(* IEC 61131-3 sources: LMM/plc, 1 file *)

(* ---- GVL.st ---- *)
VAR_GLOBAL
(* =========================================================================
   LMM 拉毛机 全局变量（唯一 GVL）
   轴：X=M1+M2，Y=M3，Z=M4，R=M5。跨距 = Y 行程（HMI_rWheelBase，4~6 m）。
   维护方式：编辑本文件后运行 tools/inject_st.py 注入 LMM.xml。
   ========================================================================= *)

(* ===== 1. 面板物理 IO（地址固定勿改） ===== *)
StartBtn AT %IX1.6 : BOOL;      (* 【面板启动】→ HMI_xStart *)
StopBtn AT %IX1.4 : BOOL;       (* 【面板停止】→ HMI_xStop *)
ResetBtn : BOOL;                (* 【面板复位】→ HMI_xStopHold3s；地址现场另绑 *)
EStop AT %IX0.4 : BOOL;         (* 【面板急停】正常=TRUE 按下=FALSE *)
StopLamp AT %QX0.6 : BOOL;      (* 【停止指示灯】← Dev_xStop *)
StartLamp AT %QX0.7 : BOOL;     (* 【运行指示灯】← Dev_xRun *)
JogFwd : BOOL;                  (* 【面板前进】手动 X+ *)
JogBwd : BOOL;                  (* 【面板后退】手动 X- *)
JogRight : BOOL;                (* 【面板右】手动 Y+ *)
JogLeft : BOOL;                 (* 【面板左】手动 Y- *)
JogUp : BOOL;                   (* 【面板上】手动 Z+ *)
JogDown : BOOL;                 (* 【面板下】手动 Z- *)
JogClockAdd : BOOL;             (* 【面板顺时针】手动 R+ *)
JogClockMis : BOOL;             (* 【面板逆时针】手动 R- *)

(* ===== 2. 安全 / 起停（PRG_TcpHmi 仲裁后写） ===== *)
HMI_xEStop : BOOL;              (* 【急停】TRUE正常 FALSE按下 = 物理 AND 触摸屏Req AND Web *)
HMI_xStop : BOOL;               (* 【停止】任一源为真即停；长按3s=复位 *)
HMI_xStopHold3s : BOOL;         (* 【复位】清急停锁存 + 轴故障复位 *)
HMI_xStart : BOOL;              (* 【启动】上升沿 *)
HMI_xEnable : BOOL;             (* 【启动别名】与 HMI_xStart 等效 *)
xEStopLatched : BOOL;           (* 【急停锁存】仅复位可清 *)
xFaultAggregate : BOOL;         (* 【故障汇总】任轴 ErrorStop *)
eCtrlSrc : INT;                 (* 【控制源】0=面板/触摸屏 1=远程Web；仅 PRG_TcpHmi 写 *)

(* ===== 3. 设备状态显示（Logic 写，只读派生，不做互锁） ===== *)
eOpMode : INT;                  (* 【运行方式】0手动 1自动 *)
iAlarmID : INT;                 (* 【内部报警号】 *)
HMI_eDevState : INT;            (* 【只读·状态码】0停 1运行 2错误 *)
HMI_eOpMode : INT;              (* 【只读·方式显示】0手动 1自动 *)
HMI_iAlarmShow : INT;           (* 【只读·报警号】1001急停 1002轴故障 1005力超时 1006从站失败 1007未就绪；1008已废 *)
Dev_xStop : BOOL;               (* 【内部·停止派生】 *)
Dev_xRun : BOOL;                (* 【内部·运行派生】 *)
Dev_xError : BOOL;              (* 【内部·故障派生】 *)
HMI_xDevStop : BOOL;            (* 【只读·停止灯】 *)
HMI_xDevRun : BOOL;             (* 【只读·运行灯】 *)
HMI_xDevError : BOOL;           (* 【只读·故障灯】 *)
HMI_xLampEStop : BOOL;          (* 【只读·急停指示】 *)
HMI_xLampEnableOk : BOOL;       (* 【只读·就绪灯】 *)
HMI_xLampFault : BOOL;          (* 【只读·故障指示】 *)

(* ===== 4. 手动点动（电平；前提：急停正常+手动+未停止） ===== *)
HMI_xAutoMode : BOOL;           (* 【模式】FALSE手动 TRUE自动 *)
HMI_xJogXPos : BOOL;            (* 【X+】M1=M2 同速同向；与旋转互斥 *)
HMI_xJogXNeg : BOOL;            (* 【X-】 *)
HMI_xSpinLeft : BOOL;           (* 【左旋转】差速原地转；与 X± 互斥 *)
HMI_xSpinRight : BOOL;          (* 【右旋转】 *)
HMI_xJogYPos : BOOL;            (* 【Y+】受限位 *)
HMI_xJogYNeg : BOOL;            (* 【Y-】 *)
HMI_xJogZPos : BOOL;            (* 【Z+】回零后软限位 [-0.7,0] *)
HMI_xJogZNeg : BOOL;            (* 【Z-】 *)
HMI_xJogRPos : BOOL;            (* 【R+】需 xM5Ready *)
HMI_xJogRNeg : BOOL;            (* 【R-】 *)
(* 点动速度 HMI_rJogVel*/rSpinVel 在 RETAIN 区 *)

(* ===== 5. 回零（上升沿；同时只回一轴） ===== *)
HMI_xHomeY : BOOL;              (* 【Y回零】 *)
HMI_xHomeZ : BOOL;              (* 【Z回零】完成后软限位生效 *)
HMI_xHomeR : BOOL;              (* 【R回零】编码器回零 *)
HMI_iHomeAxis : INT := 0;       (* 【回零轴选择】0无 1Y 2Z 3R *)
HMI_xHomeExec : BOOL;           (* 【回零执行】对选定轴 *)
HMI_xHomedY : BOOL;             (* 【只读·Y已回零】 *)
HMI_xHomedZ : BOOL;             (* 【只读·Z已回零】 *)
HMI_xHomedR : BOOL;             (* 【只读·R已回零】 *)
HMI_xHomeBusyY : BOOL;          (* 【只读·Y回零中】 *)
HMI_xHomeBusyZ : BOOL;          (* 【只读·Z回零中】 *)
HMI_xHomeBusyR : BOOL;          (* 【只读·R回零中】 *)

(* ===== 6. 自动多道循环 ===== *)
HMI_xAutoStart : BOOL;          (* 【自动启动】上升沿 *)
HMI_xAutoAbort : BOOL;          (* 【自动中止】立即结束 *)
HMI_rHeadingErr : REAL := 0.0;  (* 【航向误差】视觉/外部纠偏输入（实时量，不保持） *)
iAutoStep : INT;                (* 【自动步】0Idle..6Done *)
HMI_iAutoStepShow : INT;        (* 【只读·自动步号】 *)
HMI_xAutoBusy : BOOL;           (* 【只读·自动忙】 *)
HMI_xAutoDone : BOOL;           (* 【只读·自动完成】 *)
(* 自动参数 rAutoDistX/rAutoVel*/rWheelBase/iAutoPasses/rKp*/rForceSet 在 RETAIN 区 *)

(* ===== 7. 力控（LE 拉压传感器，组态 Modbus RTU COM0） ===== *)
Force_xEnable : BOOL := TRUE;   (* 【力通讯总使能】 *)
Force_wInRaw AT %IW102 : WORD;  (* 组态读通道：0x0000 原始力 *)
Force_wOutTare AT %QW42 : WORD; (* 组态写通道：0x0011 去皮 *)
Force_wOutUnit AT %QW43 : WORD := 5; (* 组态写通道：0x0002 单位 5=N *)
Force_rScale : REAL := 0.01;    (* 原始值倍率 *)
Force_xReadTrig : BOOL;         (* 【内部·力读触发】组态用，勿绑屏 *)
Force_xCommOk : BOOL;           (* 【只读·力通讯正常】 *)
Force_xTimeout : BOOL;          (* 【只读·力超时】报警1005 *)
Force_xSlaveFail : BOOL;        (* 【只读·从站使能失败】报警1006 *)
Force_xTareBusy : BOOL;         (* 【只读·去皮中】 *)
Force_xTareDone : BOOL;         (* 【只读·去皮完成】 *)
Force_iRaw : INT;               (* 【只读·原始计数】 *)
Force_iState : INT;             (* 【只读·力任务状态】 *)
rForceAct : REAL;               (* 【实际力】N；Axis 任务写（模拟时 Logic 写） *)
rForceKp : REAL;                (* 【内部·恒力Kp】 *)
HMI_rForceSim : REAL;           (* 【力模拟值】N *)
HMI_xForceSimEnable : BOOL;     (* 【力模拟使能】台架用 *)
HMI_xForceTare : BOOL;          (* 【去皮】上升沿 *)
HMI_xForceUntare : BOOL;        (* 【取消去皮】上升沿 *)
HMI_xForceGuide : BOOL;         (* 【力引导电平】TRUE 持续 Z 恒力跟随 *)
HMI_rForceShow : REAL;          (* 【只读·显示力】N *)
Logic_xForceTare : BOOL;        (* 【内部·自动步去皮脉冲】 *)

(* ===== 8. 硬限位配置已移至 RETAIN 区（Cfg_rLim*） ===== *)

(* ===== 9. 联锁 / 物理限位输入（地址 TBD，设备树映射） ===== *)
I_xLimYPos : BOOL;              (* 【Y正限位开关】 *)
I_xLimYNeg : BOOL;              (* 【Y负限位开关】 *)
I_xLimZPos : BOOL;              (* 【Z正限位开关】 *)
I_xLimZNeg : BOOL;              (* 【Z负限位开关】 *)
xIlk_BlockYPlus : BOOL;         (* 【联锁禁Y+】开关 ∨ Cfg 限位 *)
xIlk_BlockYNeg : BOOL;          (* 【联锁禁Y-】 *)
xIlk_BlockZPlus : BOOL;         (* 【联锁禁Z+】 *)
xIlk_BlockZNeg : BOOL;          (* 【联锁禁Z-】 *)
xM5Ready : BOOL := TRUE;        (* 【第5轴就绪】FALSE=忽略 R *)

(* ===== 10. 轴命令（Logic → Axis，仅 Logic 写） ===== *)
AxisCmd_xPower : BOOL;          (* 【轴使能】= 安全条件 *)
AxisCmd_xStopAll : BOOL;        (* 【全停】急停/停止/故障/中止 *)
AxisCmd_xResetFault : BOOL;     (* 【故障复位脉冲】 *)
AxisCmd_xJogXPos : BOOL;        (* 【X+】 *)
AxisCmd_xJogXNeg : BOOL;        (* 【X-】 *)
AxisCmd_xSpinLeft : BOOL;       (* 【左旋】 *)
AxisCmd_xSpinRight : BOOL;      (* 【右旋】 *)
AxisCmd_xJogYPos : BOOL;        (* 【Y+】 *)
AxisCmd_xJogYNeg : BOOL;        (* 【Y-】 *)
AxisCmd_xJogZPos : BOOL;        (* 【Z+】 *)
AxisCmd_xJogZNeg : BOOL;        (* 【Z-】 *)
AxisCmd_xJogRPos : BOOL;        (* 【R+】 *)
AxisCmd_xJogRNeg : BOOL;        (* 【R-】 *)
AxisCmd_xHomeY : BOOL;          (* 【Y回零】完成/停止清 *)
AxisCmd_xHomeZ : BOOL;          (* 【Z回零】 *)
AxisCmd_xHomeR : BOOL;          (* 【R回零】 *)
AxisCmd_xMoveRelX : BOOL;       (* 【X相对走距】速度模式+里程判完成 *)
AxisCmd_rMoveDistX : REAL;      (* 【X相对距离】 *)
AxisCmd_rMoveVelX : REAL;       (* 【X相对速度】 *)
AxisCmd_xMoveRelY : BOOL;       (* 【Y相对】 *)
AxisCmd_rMoveDistY : REAL;      (* 【Y相对距离】自动=跨距 *)
AxisCmd_rMoveVelY : REAL;       (* 【Y速度】 *)
AxisCmd_xMoveAbsY : BOOL;       (* 【Y绝对】归位用 *)
AxisCmd_rMoveAbsPosY : REAL;    (* 【Y绝对目标】 *)
AxisCmd_xForceFollow : BOOL;    (* 【Z力跟随】 *)
AxisCmd_rForceSet : REAL;       (* 【力目标】 *)
AxisCmd_rForceKp : REAL;        (* 【力Kp】 *)
AxisCmd_rForceVelMax : REAL;    (* 【力跟随限速】 *)
AxisCmd_xHoldR : BOOL;          (* 【R保持角】 *)
AxisCmd_rRHoldPos : REAL;       (* 【R保持角位置】 *)
AxisCmd_rHeadingErr : REAL;     (* 【航向误差】 *)
AxisCmd_rTrackKp : REAL;        (* 【纠偏Kp】 *)
AxisCmd_rJogVelX : REAL;        (* 【X点动速度】 *)
AxisCmd_rSpinVel : REAL := 0.0; (* 【旋转速度】 *)
AxisCmd_rJogVelY : REAL;        (* 【Y点动速度】 *)
AxisCmd_rJogVelZ : REAL;        (* 【Z点动速度】 *)
AxisCmd_rJogVelR : REAL;        (* 【R点动速度】 *)
AxisCmd_rWheelBase : REAL;      (* 【跨距】限幅 4..6 *)
AxisCmd_rAccX : REAL;           (* 【X加速度】 *)
AxisCmd_rDecX : REAL;           (* 【X减速度】 *)
AxisCmd_rAccY : REAL;           (* 【Y加速度】 *)
AxisCmd_rDecY : REAL;           (* 【Y减速度】 *)
AxisCmd_rAccZ : REAL;           (* 【Z加速度】 *)
AxisCmd_rDecZ : REAL;           (* 【Z减速度】 *)
AxisCmd_rAccR : REAL;           (* 【R加速度】 *)
AxisCmd_rDecR : REAL;           (* 【R减速度】 *)

(* ===== 11. 轴反馈（Axis → Logic，仅 Axis 任务写） ===== *)
AxisFb_rVelCmdM1 : REAL;        (* 【只读·M1速度指令】含纠偏/旋转 *)
AxisFb_rVelCmdM2 : REAL;        (* 【只读·M2速度指令】 *)
AxisFb_rPosM1 : REAL;           (* 【只读·M1位置】 *)
AxisFb_rPosM2 : REAL;           (* 【只读·M2位置】 *)
AxisFb_rPosX : REAL;            (* 【只读·Virtual X 位置】走距判据 *)
AxisFb_rSyncErr : REAL;         (* 【只读·M1-M2 同步误差】 *)
AxisFb_rVelFactorX : REAL;      (* 【只读·Virtual Override 倍率】 *)
AxisFb_xGantryCoupled : BOOL;   (* 【只读·龙门已 GearIn】M1且M2 *)
AxisFb_xInGearM1 : BOOL;        (* 【只读·M1 电子齿轮 InGear】 *)
AxisFb_xInGearM2 : BOOL;        (* 【只读·M2 电子齿轮 InGear】 *)
AxisFb_xPoweredV : BOOL;        (* 【只读·Virtual 已使能】 *)
AxisFb_xSyncWarn : BOOL;        (* 【只读·同步预警】 *)
AxisFb_xSyncFault : BOOL;       (* 【只读·同步跳闸】已废，恒 FALSE *)
AxisFb_iGantryState : INT;      (* 【只读·0Idle 1Coupling 2Coupled 3Decouple 4Diff 5Align】 *)
AxisFb_rPosY : REAL;            (* 【只读·Y位置】 *)
AxisFb_rPosZ : REAL;            (* 【只读·Z位置】 *)
AxisFb_rPosR : REAL;            (* 【只读·R位置/角度】 *)
AxisFb_xStandstill1 : BOOL;     (* 【只读·M1静止】 *)
AxisFb_xStandstill2 : BOOL;     (* 【只读·M2静止】 *)
AxisFb_xStandstillY : BOOL;     (* 【只读·Y静止】 *)
AxisFb_xStandstillZ : BOOL;     (* 【只读·Z静止】 *)
AxisFb_xStandstillR : BOOL;     (* 【只读·R静止】 *)
AxisFb_xMovingM1 : BOOL;        (* 【只读·M1运动中】 *)
AxisFb_xMovingM2 : BOOL;        (* 【只读·M2运动中】 *)
AxisFb_xMovingY : BOOL;         (* 【只读·Y运动中】 *)
AxisFb_xMovingZ : BOOL;         (* 【只读·Z运动中】 *)
AxisFb_xMovingR : BOOL;         (* 【只读·R运动中】 *)
AxisFb_xPoweredM1 : BOOL;       (* 【只读·M1已使能】 *)
AxisFb_xPoweredM2 : BOOL;       (* 【只读·M2已使能】 *)
AxisFb_xPoweredY : BOOL;        (* 【只读·Y已使能】 *)
AxisFb_xPoweredZ : BOOL;        (* 【只读·Z已使能】 *)
AxisFb_xPoweredR : BOOL;        (* 【只读·R已使能】 *)
AxisFb_xReadyM1 : BOOL;         (* 【只读·M1就绪】 *)
AxisFb_xReadyM2 : BOOL;         (* 【只读·M2就绪】 *)
AxisFb_xReadyY : BOOL;          (* 【只读·Y就绪】 *)
AxisFb_xReadyZ : BOOL;          (* 【只读·Z就绪】 *)
AxisFb_xReadyR : BOOL;          (* 【只读·R就绪】 *)
AxisFb_xReady : BOOL;           (* 【只读·全轴就绪】FALSE → 报警1007 *)
AxisFb_xHomedY : BOOL;          (* 【只读·Y已回零】 *)
AxisFb_xHomedZ : BOOL;          (* 【只读·Z已回零】 *)
AxisFb_xHomedR : BOOL;          (* 【只读·R已回零】 *)
AxisFb_xFaultM1 : BOOL;         (* 【只读·M1故障】 *)
AxisFb_xFaultM2 : BOOL;         (* 【只读·M2故障】 *)
AxisFb_xFaultY : BOOL;          (* 【只读·Y故障】 *)
AxisFb_xFaultZ : BOOL;          (* 【只读·Z故障】 *)
AxisFb_xFaultR : BOOL;          (* 【只读·R故障】 *)
AxisFb_xMoveDoneX : BOOL;       (* 【只读·X走距完成】 *)
AxisFb_xMoveDoneY : BOOL;       (* 【只读·Y完成】 *)

(* ===== 12. Modbus 过程映像 + Web 影子（仅 PRG_TcpHmi 写） ===== *)
MB_CmdIn AT %IW103 : ARRAY[0..95] OF WORD;   (* 【命令入】Holding 1000..1095 *)
MB_StatusOut AT %QW44 : ARRAY[0..95] OF WORD;(* 【状态出】Holding 1100..1195 *)
Tcp_iCommStatus : INT;          (* 【只读·通讯诊断】0离线 1在线 2版本错 3序号错 4超时 *)
Tcp_xConnected : BOOL;          (* 【只读·远程已连接】 *)
Tcp_xTimeout : BOOL;            (* 【只读·远程超时】 *)
Tcp_xOnline : BOOL;             (* 【只读·远程在线可用】 *)
Tcp_wLastHb : WORD;             (* 【内部·上次心跳】 *)
Tcp_wLastSeq : WORD;            (* 【内部·上次命令序号】 *)
Tcp_wStatusSeq : WORD;          (* 【内部·状态序号】 *)
Tcp_xEStop : BOOL := TRUE;      (* 【Web影子·急停】掉线强制 TRUE *)
Tcp_xStop : BOOL;               (* 【Web影子·停止】 *)
Tcp_xStopHold3s : BOOL;         (* 【Web影子·复位】 *)
Tcp_xStart : BOOL;              (* 【Web影子·启动】 *)
Tcp_xEnable : BOOL;             (* 【Web影子·启动别名】 *)
Tcp_xAutoMode : BOOL;           (* 【Web影子·模式】 *)
Tcp_xJogXPos : BOOL;            (* 【Web影子·X+】 *)
Tcp_xJogXNeg : BOOL;            (* 【Web影子·X-】 *)
Tcp_xSpinLeft : BOOL;           (* 【Web影子·左旋】 *)
Tcp_xSpinRight : BOOL;          (* 【Web影子·右旋】 *)
Tcp_xJogYPos : BOOL;            (* 【Web影子·Y+】 *)
Tcp_xJogYNeg : BOOL;            (* 【Web影子·Y-】 *)
Tcp_xJogZPos : BOOL;            (* 【Web影子·Z+】 *)
Tcp_xJogZNeg : BOOL;            (* 【Web影子·Z-】 *)
Tcp_xJogRPos : BOOL;            (* 【Web影子·R+】 *)
Tcp_xJogRNeg : BOOL;            (* 【Web影子·R-】 *)
Tcp_xHomeY : BOOL;              (* 【Web影子·Y回零】 *)
Tcp_xHomeZ : BOOL;              (* 【Web影子·Z回零】 *)
Tcp_xHomeR : BOOL;              (* 【Web影子·R回零】 *)
Tcp_iHomeAxis : INT := 0;       (* 【Web影子·回零轴选择】 *)
Tcp_xHomeExec : BOOL;           (* 【Web影子·回零执行】 *)
Tcp_rJogVelX : REAL := 0.4;     (* 【Web影子·X速度】 *)
Tcp_rSpinVel : REAL := 0.3;     (* 【Web影子·旋转速度】 *)
Tcp_rJogVelY : REAL := 0.3;     (* 【Web影子·Y速度】 *)
Tcp_rJogVelZ : REAL := 0.2;     (* 【Web影子·Z速度】 *)
Tcp_rJogVelR : REAL := 0.2;     (* 【Web影子·R速度】 *)
Tcp_xAutoStart : BOOL;          (* 【Web影子·自动启动】 *)
Tcp_xAutoAbort : BOOL;          (* 【Web影子·自动中止】 *)
Tcp_rAutoDistX : REAL := 1.0;   (* 【Web影子·自动X距】 *)
Tcp_rAutoVelX : REAL := 0.4;    (* 【Web影子·自动X速】 *)
Tcp_rAutoVelY : REAL := 0.3;    (* 【Web影子·自动Y速】 *)
Tcp_rAutoVelZ : REAL := 0.15;   (* 【Web影子·自动Z速】 *)
Tcp_rWheelBase : REAL := 5.0;   (* 【Web影子·跨距】 *)
Tcp_rForceSet : REAL := 100.0;  (* 【Web影子·力设定】 *)
Tcp_xForceSimEnable : BOOL := FALSE; (* 【Web影子·力模拟使能】 *)
Tcp_rForceSim : REAL;           (* 【Web影子·力模拟值】 *)
Tcp_xForceTare : BOOL;          (* 【Web影子·去皮】 *)
Tcp_xForceUntare : BOOL;        (* 【Web影子·取消去皮】 *)
Tcp_xForceGuide : BOOL;         (* 【Web影子·力引导】 *)
Tcp_iAutoPasses : INT := 1;     (* 【Web影子·自动道数】 *)
Tcp_rHeadingErr : REAL := 0.0;  (* 【Web影子·航向误差】 *)
Tcp_rKpTrack : REAL;            (* 【Web影子·纠偏Kp】 *)
Tcp_rKpForce : REAL;            (* 【Web影子·力Kp】 *)
Tcp_rAccX : REAL := 100.0;      (* 【Web影子·X加速度】 *)
Tcp_rDecX : REAL := 100.0;      (* 【Web影子·X减速度】 *)
Tcp_rAccY : REAL := 100.0;      (* 【Web影子·Y加速度】 *)
Tcp_rDecY : REAL := 100.0;      (* 【Web影子·Y减速度】 *)
Tcp_rAccZ : REAL := 100.0;      (* 【Web影子·Z加速度】 *)
Tcp_rDecZ : REAL := 100.0;      (* 【Web影子·Z减速度】 *)
Tcp_rAccR : REAL := 100.0;      (* 【Web影子·R加速度】 *)
Tcp_rDecR : REAL := 100.0;      (* 【Web影子·R减速度】 *)

(* ===== 13. 触摸屏请求（仅触摸屏写；PRG_TcpHmi 仲裁并入，防双写自锁） ===== *)
HMI_xStartReq : BOOL;           (* 【触摸屏启动】 *)
HMI_xStopReq : BOOL;            (* 【触摸屏停止】 *)
HMI_xResetReq : BOOL;           (* 【触摸屏复位】 *)
HMI_xEStopReq : BOOL := TRUE;   (* 【触摸屏急停】TRUE正常 *)
HMI_xAutoStartReq : BOOL;       (* 【触摸屏自动启动】 *)
HMI_xAutoAbortReq : BOOL;       (* 【触摸屏自动中止】 *)
END_VAR

VAR_GLOBAL RETAIN
(* =========================================================================
   掉电保存参数（HMI/触摸屏/Web 可改，断电保持）
   注入时并入唯一 GVL（InoPro 每个 globalvars data 仅允许一个 globalVars），
   变量带 retain 属性；勿再拆成 GVL_RETAIN 兄弟节点。
   ========================================================================= *)

(* ===== R1. 每轴点动速度 ===== *)
HMI_rJogVelX : REAL := 0.4;     (* 【X直行速度】与旋转速度分开 *)
HMI_rSpinVel : REAL := 0.3;     (* 【左右旋速度】 *)
HMI_rJogVelY : REAL := 0.4;     (* 【Y点动速度】 *)
HMI_rJogVelZ : REAL := 0.4;     (* 【Z点动速度】力跟随限速后备 *)
HMI_rJogVelR : REAL := 0.2;     (* 【R点动速度】 *)

(* ===== R2. 每轴加减速（<1 时 Logic 取 100） ===== *)
HMI_rAccX : REAL := 100.0;      (* 【X加速度】 *)
HMI_rDecX : REAL := 100.0;      (* 【X减速度】 *)
HMI_rAccY : REAL := 100.0;      (* 【Y加速度】 *)
HMI_rDecY : REAL := 100.0;      (* 【Y减速度】 *)
HMI_rAccZ : REAL := 100.0;      (* 【Z加速度】 *)
HMI_rDecZ : REAL := 100.0;      (* 【Z减速度】 *)
HMI_rAccR : REAL := 100.0;      (* 【R加速度】 *)
HMI_rDecR : REAL := 100.0;      (* 【R减速度】 *)

(* ===== R3. 自动工艺参数 ===== *)
HMI_rAutoDistX : REAL := 1.0;   (* 【自动X走距】每道 *)
HMI_rAutoVelX : REAL := 0.4;    (* 【自动X速度】 *)
HMI_rAutoVelY : REAL := 0.3;    (* 【自动Y速度】 *)
HMI_rAutoVelZ : REAL := 0.15;   (* 【自动Z速度】力跟随限速参考 *)
HMI_rWheelBase : REAL := 5.0;   (* 【龙门跨距=Y行程】4~6 m *)
HMI_iAutoPasses : INT := 1;     (* 【自动总道数】≥1 *)
HMI_rForceSet : REAL := 100.0;  (* 【恒力设定】N *)
HMI_rKpForce : REAL := 1.0;     (* 【力跟随Kp】 *)
HMI_rKpTrack : REAL := 0.0;     (* 【直线纠偏Kp】 *)

(* ===== R4. 硬限位配置（X 无；所有模式强制，FB_Servo 执行） ===== *)
Cfg_rLimYPos : REAL := 6.0;     (* 【Y正限位】m，默认跨距上限 *)
Cfg_rLimYNeg : REAL := 0.0;     (* 【Y负限位】m *)
Cfg_rLimZPos : REAL := 0.0;     (* 【Z正限位】上 *)
Cfg_rLimZNeg : REAL := -0.7;    (* 【Z负限位】下压行程 *)
Cfg_rLimRPos : REAL := 180.0;   (* 【R正限位】度 *)
Cfg_rLimRNeg : REAL := -180.0;  (* 【R负限位】度 *)

(* ===== R5. X 龙门同步 / Override / 跟轨 ===== *)
Cfg_rVelBaseMaxX : REAL := 1.0; (* 【X速度基准】诊断倍率分母；≥最大 Jog/Auto *)
Cfg_rPhaseMax : REAL := 0.01;   (* 【跟轨相位限幅】u；连续 Phasing *)
Cfg_rSyncWarn : REAL := 0.02;   (* 【同步预警】|M1-M2|；降速 *)
Cfg_rSyncFault : REAL := 0.05;  (* 【同步跳闸】已废；保留 RETAIN 布局 *)
END_VAR

VAR_GLOBAL
(* ===== R6. G 线视觉/Web 单轴直控（0.60 X 双电机，0.68 全轴；唯一写者见注释） ===== *)
HMI_xDirectEnable : BOOL;       (* 【X直控·Web使能】命令镜像 word5 bit10；与 Vis_xEnable 取或 *)
HMI_rVelM1Set : REAL;           (* 【X直控·M1设定速度】m/s；命令镜像 word54 ×1000 *)
HMI_rVelM2Set : REAL;           (* 【X直控·M2设定速度】m/s；命令镜像 word55 ×1000 *)
Vis_xEnable : BOOL;             (* 【视觉直控使能】命令 word56 bit0；网关中继写 *)
Vis_wSeq : WORD;                (* 【视觉心跳序号】命令 word57 *)
Vis_rVelM1Set : REAL;           (* 【视觉直控·M1速度】命令 word58 ×1000 *)
Vis_rVelM2Set : REAL;           (* 【视觉直控·M2速度】命令 word59 ×1000 *)
Direct_xActive : BOOL;          (* 【只读·X直控·FB在役】Axis 任务写；状态 word28 bit0 *)
Direct_xOnline : BOOL;          (* 【只读·X直控·视觉在线】Logic 写；状态 word28 bit1 *)
Direct_xEnable : BOOL;          (* 【只读·X直控·仲裁后使能】Logic 写；状态 word28 bit2 *)
Direct_rVelM1Act : REAL;        (* 【只读·X直控·M1实际速度】Axis 任务写；状态 word29 ×1000 *)
Direct_rVelM2Act : REAL;        (* 【只读·X直控·M2实际速度】Axis 任务写；状态 word30 ×1000 *)
Direct_wSeqEcho : WORD;         (* 【只读·X直控·视觉序号回显】Logic 写；状态 word31 *)
AxisFb_rVelActM1 : REAL;        (* 【只读·M1实际速度】Axis 任务写；状态 word32/33 ×1000；仅 Axis 任务写 *)
AxisFb_rVelActM2 : REAL;        (* 【只读·M2实际速度】Axis 任务写；状态 word34/35 ×1000；仅 Axis 任务写 *)
AxisCmd_xDirectVel : BOOL;      (* 【X直控·命令】Logic→Axis：FB_XDual 走 eMode=4 外部直控 *)
AxisCmd_rVelM1Set : REAL;       (* 【X直控·M1目标速度】m/s；仅 Logic 写 *)
AxisCmd_rVelM2Set : REAL;       (* 【X直控·M2目标速度】m/s；仅 Logic 写 *)

(* ===== R7. 全轴直控命令镜像（0.68；视觉与操作员共用 word60..75，PRG_TcpHmi 写） ===== *)
HMI_iDirectModeX : UINT;        (* 【直控·X模式】命令 word60；0idle 1vel（X 仅速度） *)
HMI_rDirectPosX : REAL;         (* 【直控·X整机目标位置】命令 word61/62 ×1000；整机速度环可选 *)
HMI_iDirectModeY : UINT;        (* 【直控·Y模式】命令 word63；0idle 1vel 2posAbs 3posRel *)
HMI_rDirectVelY : REAL;         (* 【直控·Y速度】命令 word64 ×1000；m/s *)
HMI_rDirectPosY : REAL;         (* 【直控·Y目标位置】命令 word65/66 ×1000；m *)
HMI_iDirectModeZ : UINT;        (* 【直控·Z模式】命令 word67；0idle 1vel 2posAbs 3posRel *)
HMI_rDirectVelZ : REAL;         (* 【直控·Z速度】命令 word68 ×1000；m/s *)
HMI_rDirectPosZ : REAL;         (* 【直控·Z目标位置】命令 word69/70 ×1000；m *)
HMI_iDirectModeR : UINT;        (* 【直控·R模式】命令 word71；0idle 1vel 2posAbs 3posRel *)
HMI_rDirectVelR : REAL;         (* 【直控·R速度】命令 word72 ×1000；工程单位/s *)
HMI_rDirectPosR : REAL;         (* 【直控·R目标位置】命令 word73/74 ×1000；工程单位 *)
HMI_wDirectSeq : WORD;          (* 【直控·心跳序号】命令 word75；300ms 不变退出直控 *)
Direct2_xActiveX : BOOL;        (* 【只读·直控·X在役】Logic 写；状态 word42 bit0 *)
Direct2_xActiveY : BOOL;        (* 【只读·直控·Y在役】Logic 写；状态 word42 bit1 *)
Direct2_xActiveZ : BOOL;        (* 【只读·直控·Z在役】Logic 写；状态 word42 bit2 *)
Direct2_xActiveR : BOOL;        (* 【只读·直控·R在役】Logic 写；状态 word42 bit3 *)
Direct2_xOnline : BOOL;         (* 【只读·直控·心跳在线】Logic 写；状态 word42 bit4 *)
Direct2_xSafe : BOOL;           (* 【只读·直控·安全允许】Logic 写；状态 word42 bit5 *)
Direct2_wSeqEcho : WORD;        (* 【只读·直控·心跳回显】Logic 写；状态 word43 *)
HMI_rForceSetEcho : REAL;       (* 【只读·力设定回显】Logic 写；状态 word44/45 ×100 *)
AxisFb_rVelActY : REAL;         (* 【只读·Y实际速度】Axis 任务写；状态 word39 ×1000；仅 Axis 任务写 *)
AxisFb_rVelActZ : REAL;         (* 【只读·Z实际速度】Axis 任务写；状态 word40 ×1000；仅 Axis 任务写 *)
AxisFb_rVelActR : REAL;         (* 【只读·R实际速度】Axis 任务写；状态 word41 ×1000；仅 Axis 任务写 *)
AxisCmd_xDirectVelY : BOOL;     (* 【直控·Y速度命令】仅 Logic 写 *)
AxisCmd_rDirectVelY : REAL;     (* 【直控·Y进给速度】m/s；模式 1 速度，2/3 定位限速 *)
AxisCmd_xDirectAbsY : BOOL;     (* 【直控·Y绝对命令】仅 Logic 写 *)
AxisCmd_rDirectAbsY : REAL;     (* 【直控·Y绝对目标】已钳位软限位 *)
AxisCmd_xDirectRelY : BOOL;     (* 【直控·Y相对命令】仅 Logic 写 *)
AxisCmd_rDirectRelY : REAL;     (* 【直控·Y相对距离】FB_Servo 内钳位 *)
AxisCmd_xDirectVelZ : BOOL;     (* 【直控·Z速度命令】仅 Logic 写 *)
AxisCmd_rDirectVelZ : REAL;     (* 【直控·Z进给速度】m/s *)
AxisCmd_xDirectAbsZ : BOOL;     (* 【直控·Z绝对命令】仅 Logic 写 *)
AxisCmd_rDirectAbsZ : REAL;     (* 【直控·Z绝对目标】已钳位软限位 *)
AxisCmd_xDirectRelZ : BOOL;     (* 【直控·Z相对命令】仅 Logic 写 *)
AxisCmd_rDirectRelZ : REAL;     (* 【直控·Z相对距离】FB_Servo 内钳位 *)
AxisCmd_xDirectVelR : BOOL;     (* 【直控·R速度命令】仅 Logic 写 *)
AxisCmd_rDirectVelR : REAL;     (* 【直控·R进给速度】工程单位/s *)
AxisCmd_xDirectAbsR : BOOL;     (* 【直控·R绝对命令】仅 Logic 写 *)
AxisCmd_rDirectAbsR : REAL;     (* 【直控·R绝对目标】已钳位软限位 *)
AxisCmd_xDirectRelR : BOOL;     (* 【直控·R相对命令】仅 Logic 写 *)
AxisCmd_rDirectRelR : REAL;     (* 【直控·R相对距离】FB_Servo 内钳位 *)

(* ===== R7b. 全轴直控命令影子（0.68；仅 PRG_TcpHmi 解码写，仲裁后写 HMI_*） ===== *)
Tcp_iDirectModeX : UINT;        (* 【影子·X模式】word60 *)
Tcp_rDirectPosX : REAL;         (* 【影子·X整机目标】word61/62 ×1000 *)
Tcp_iDirectModeY : UINT;        (* 【影子·Y模式】word63 *)
Tcp_rDirectVelY : REAL;         (* 【影子·Y速度】word64 ×1000 *)
Tcp_rDirectPosY : REAL;         (* 【影子·Y目标】word65/66 ×1000 *)
Tcp_iDirectModeZ : UINT;        (* 【影子·Z模式】word67 *)
Tcp_rDirectVelZ : REAL;         (* 【影子·Z速度】word68 ×1000 *)
Tcp_rDirectPosZ : REAL;         (* 【影子·Z目标】word69/70 ×1000 *)
Tcp_iDirectModeR : UINT;        (* 【影子·R模式】word71 *)
Tcp_rDirectVelR : REAL;         (* 【影子·R速度】word72 ×1000 *)
Tcp_rDirectPosR : REAL;         (* 【影子·R目标】word73/74 ×1000 *)
Tcp_wDirectSeq : WORD;          (* 【影子·直控心跳】word75 *)
END_VAR

VAR_GLOBAL RETAIN
(* ===== R8. 全轴直控配置（0.68，掉电保持） ===== *)
Cfg_rDirectVelMaxX : REAL := 0.5;  (* 【直控速度上限·X】m/s *)
Cfg_rDirectVelMaxY : REAL := 0.5;  (* 【直控速度上限·Y】m/s *)
Cfg_rDirectVelMaxZ : REAL := 0.2;  (* 【直控速度上限·Z】m/s *)
Cfg_rDirectVelMaxR : REAL := 30.0; (* 【直控速度上限·R】工程单位/s *)
Cfg_tDirectTimeout : TIME := T#300MS; (* 【直控看门狗】HMI_wDirectSeq 不变即退出 *)
END_VAR
